{attribute 'OPC.UA.DA.StructuredType' := '1'}
TYPE ST_ActiveWallModulesSetParameters :
STRUCT
	bHeatingModeAlgorithm : BOOL;
	bHeatingModeManual : BOOL;
	nControlModeAlgorithm : E_ActiveWallModulesControlMode;
	nControlModeManual : E_ActiveWallModulesControlMode;
	fHysteresisRangeAlgorithm : REAL;
	fHysteresisRangeManual : REAL; 
END_STRUCT
END_TYPE

(* stored: Version 1.1.0.1, ProductVersion 3.1.4024.6
   DUT ST_ActiveWallModulesSetParameters: Id {10529f76-ffb1-4fa2-964c-d8ab4c4354c2} *)
